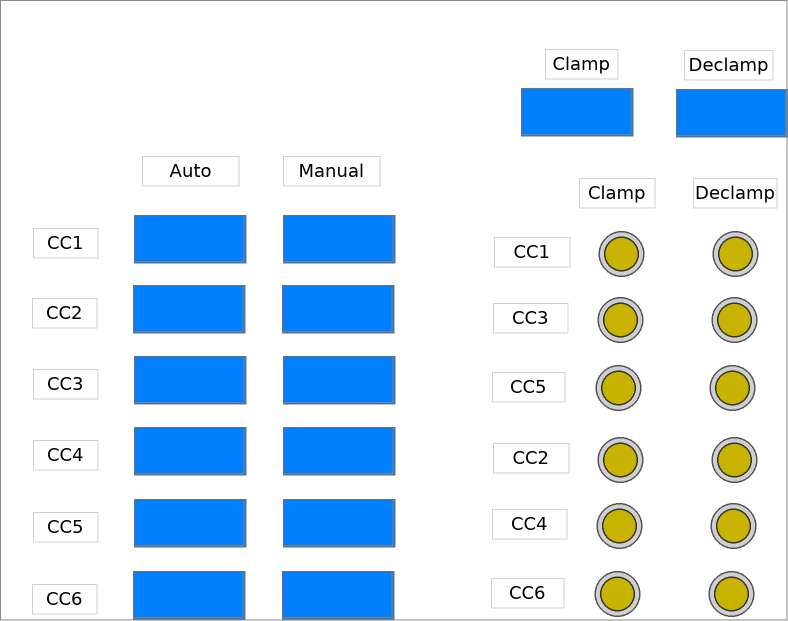
VISUALIZATION Manual_Action_Fix2  // 788x621
    Textfield (142,156 97x30), "Auto"
    Textfield (545,49 73x30), "Clamp"
    Button (521,88 112x48)
        p573394764: Auto_Cycle_Fix2.Fixture_2.Unit_Adv_Pb
        tap Auto_Cycle_Fix2.Fixture_2.Unit_Adv_Pb
    Textfield (684,50 89x30), "Declamp"
    Button (676,89 112x48)
        p573394764: Auto_Cycle_Fix2.Fixture_2.Unit_Ret_Pb
        tap Auto_Cycle_Fix2.Fixture_2.Unit_Ret_Pb
    Textfield (494,237 76x30), "CC1"
    Textfield (493,303 75x30), "CC3"
    Textfield (492,372 73x30), "CC5"
    Lamp1 (595,227 53x54), variable: Auto_Cycle_Fix2.Fixture_2.CC1_Output.Work_Position, style: Lamp-Lamp1-Yellow
    Lamp1 (594,293 53x54), variable: Auto_Cycle_Fix2.Fixture_2.CC3_Output.Work_Position, style: Lamp-Lamp1-Yellow
    Lamp1 (592,361 53x54), variable: Auto_Cycle_Fix2.Fixture_2.CC5_Output.Work_Position, style: Lamp-Lamp1-Yellow
    Textfield (579,178 76x30), "Clamp"
    Lamp1 (709,227 53x54), variable: Auto_Cycle_Fix2.Fixture_2.CC1_Output.Home_Position, style: Lamp-Lamp1-Yellow
    Lamp1 (708,293 53x54), variable: Auto_Cycle_Fix2.Fixture_2.CC3_Output.Home_Position, style: Lamp-Lamp1-Yellow
    Lamp1 (706,361 53x54), variable: Auto_Cycle_Fix2.Fixture_2.CC5_Output.Home_Position, style: Lamp-Lamp1-Yellow
    Textfield (693,178 84x30), "Declamp"
    Textfield (493,443 76x30), "CC2"
    Textfield (492,509 75x30), "CC4"
    Textfield (491,578 73x30), "CC6"
    Lamp1 (594,433 53x54), variable: Auto_Cycle_Fix2.Fixture_2.CC2_Output.Work_Position, style: Lamp-Lamp1-Yellow
    Lamp1 (593,499 53x54), variable: Auto_Cycle_Fix2.Fixture_2.CC4_Output.Work_Position, style: Lamp-Lamp1-Yellow
    Lamp1 (591,567 53x54), variable: Auto_Cycle_Fix2.Fixture_2.CC6_Output.Work_Position, style: Lamp-Lamp1-Yellow
    Lamp1 (708,433 53x54), variable: Auto_Cycle_Fix2.Fixture_2.CC2_Output.Home_Position, style: Lamp-Lamp1-Yellow
    Lamp1 (707,499 53x54), variable: Auto_Cycle_Fix2.Fixture_2.CC4_Output.Home_Position, style: Lamp-Lamp1-Yellow
    Lamp1 (705,567 53x54), variable: Auto_Cycle_Fix2.Fixture_2.CC6_Output.Home_Position, style: Lamp-Lamp1-Yellow
    Button (134,215 112x48)
        p573394764: Auto_Cycle_Fix2.Fixture_2.CC1_Input.Auto_Sel
        toggle Auto_Cycle_Fix2.Fixture_2.CC1_Input.Auto_Sel
    Textfield (33,228 65x30), "CC1"
    Button (133,285 112x48)
        p573394764: Auto_Cycle_Fix2.Fixture_2.CC2_Input.Auto_Sel
        toggle Auto_Cycle_Fix2.Fixture_2.CC2_Input.Auto_Sel
    Textfield (32,298 65x30), "CC2"
    Button (134,356 112x48)
        p573394764: Auto_Cycle_Fix2.Fixture_2.CC3_Input.Auto_Sel
        toggle Auto_Cycle_Fix2.Fixture_2.CC3_Input.Auto_Sel
    Textfield (33,369 65x30), "CC3"
    Button (134,427 112x48)
        p573394764: Auto_Cycle_Fix2.Fixture_2.CC4_Input.Auto_Sel
        toggle Auto_Cycle_Fix2.Fixture_2.CC4_Input.Auto_Sel
    Textfield (33,440 65x30), "CC4"
    Button (134,499 112x48)
        p573394764: Auto_Cycle_Fix2.Fixture_2.CC5_Input.Auto_Sel
        toggle Auto_Cycle_Fix2.Fixture_2.CC5_Input.Auto_Sel
    Textfield (33,512 65x30), "CC5"
    Button (133,571 112x48)
        p573394764: Auto_Cycle_Fix2.Fixture_2.CC6_Input.Auto_Sel
        toggle Auto_Cycle_Fix2.Fixture_2.CC6_Input.Auto_Sel
    Textfield (32,584 65x30), "CC6"
    Button (283,215 112x48)
        p573394764: Auto_Cycle_Fix2.Fixture_2.CC1_Input.Manual_Sel
        toggle Auto_Cycle_Fix2.Fixture_2.CC1_Input.Manual_Sel
    Button (282,285 112x48)
        p573394764: Auto_Cycle_Fix2.Fixture_2.CC2_Input.Manual_Sel
        toggle Auto_Cycle_Fix2.Fixture_2.CC2_Input.Manual_Sel
    Button (283,356 112x48)
        p573394764: Auto_Cycle_Fix2.Fixture_2.CC3_Input.Manual_Sel
        toggle Auto_Cycle_Fix2.Fixture_2.CC3_Input.Manual_Sel
    Button (283,427 112x48)
        p573394764: Auto_Cycle_Fix2.Fixture_2.CC4_Input.Manual_Sel
        toggle Auto_Cycle_Fix2.Fixture_2.CC4_Input.Manual_Sel
    Button (283,499 112x48)
        p573394764: Auto_Cycle_Fix2.Fixture_2.CC5_Input.Manual_Sel
        toggle Auto_Cycle_Fix2.Fixture_2.CC5_Input.Manual_Sel
    Button (282,571 112x48)
        p573394764: Auto_Cycle_Fix2.Fixture_2.CC6_Input.Manual_Sel
        toggle Auto_Cycle_Fix2.Fixture_2.CC6_Input.Manual_Sel
    Textfield (283,156 97x30), "Manual"
END_VISUALIZATION

(* stored: Version 1.1.0.1, ProductVersion 3.1.4024.16
   Visu Manual_Action_Fix2: Id {d0045204-5ccf-4ca5-b1ea-63b392d0dfc7} *)
